// TIA Portal project "taglierina_V15.1" (V15.1)

(* hardware
DEVICE "S71500/ET200MP station_1"  S7-1500 station
   slot 0: "Telaio di montaggio_0"  Rack  6ES7 590-1***0-0AA0
   slot 0: "PM 190W 120/230VAC"  PM 190W 120/230VAC  6EP1333-4BA00
   slot 1: "PLC_1"  CPU 1516-3 PN/DP  6ES7 516-3AN01-0AB0  V2.5
      slot 3: "Display CPU_1"  6ES7591-1BA00-0AA0
   slot 2: "DI 32x24VDC HF_1"  DI 32x24VDC HF  6ES7 521-1BL00-0AB0  V2.0
   slot 3: "DQ 32x24VDC/0.5A HF_1"  DQ 32x24VDC/0.5A HF  6ES7 522-1BL01-0AB0  V1.0
   slot 4: "AI 8xU/I/RTD/TC ST_1"  AI 8xU/I/RTD/TC ST  6ES7 531-7KF00-0AB0  V2.0
   slot 5: "AQ 4xU/I ST_1"  AQ 4xU/I ST  6ES7 532-5HD00-0AB0  V2.0
*)

// ===== PLC "PLC_1"  CPU 1516-3 PN/DP =====

VAR_GLOBAL   // PLC tag table "Tabella delle variabili standard"
   "Clock_Byte" AT %MB100 : Byte;
   "Clock_10Hz" AT %M100.0 : Bool;
   "Clock_5Hz" AT %M100.1 : Bool;
   "Clock_2.5Hz" AT %M100.2 : Bool;
   "Clock_2Hz" AT %M100.3 : Bool;
   "Clock_1.25Hz" AT %M100.4 : Bool;
   "Clock_1Hz" AT %M100.5 : Bool;
   "Clock_0.625Hz" AT %M100.6 : Bool;
   "Clock_0.5Hz" AT %M100.7 : Bool;
   "tmp" AT %M99.0 : Bool;
   "iApriMorsa" AT %I0.0 : Bool;   // Pulsante Morsa aperta
   "iChiudiMorsa" AT %I0.1 : Bool;   // Pulsante Morsa chiusa
   "iAuto" AT %I0.2 : Bool;   // Pulsante Marcia
   "iReset" AT %I0.3 : Bool;   // Pulsante Inizializzazione
   "iStop" AT %I0.4 : Bool;   // Pulsante Stop
   "iIndietro" AT %I0.5 : Bool;   // Taglierina in sede
   "iAvanti" AT %I0.6 : Bool;   // Taglierina Fuori Sede
   "tag_1" AT %I0.7 : Bool;
   "iMorsa2Far" AT %I1.0 : Bool;   // Morsa Mobile Lontana
   "tag_2" AT %I1.1 : Bool;
   "iMorsa1Ch" AT %I1.2 : Bool;   // Morsa Fissa Chiusa (Logica Negata)
   "tag_3" AT %I1.3 : Bool;
   "iMorsa2Ch" AT %I1.4 : Bool;   // Morsa Mobile Chiusa (Logica Negata)
   "iSchermo" AT %I1.5 : Bool;   // Sensore Schermo Sicurezza
   "iEmergenza" AT %I1.6 : Bool;   // Pulsante Emergenza (NC)
   "Tag_16" AT %I1.7 : Bool;
   "Tag_17" AT %I2.0 : Bool;
   "Tag_18" AT %I2.1 : Bool;
   "Tag_19" AT %I2.2 : Bool;
   "Tag_20" AT %I2.3 : Bool;
   "Tag_21" AT %I2.4 : Bool;
   "Tag_22" AT %I2.5 : Bool;
   "Tag_23" AT %I2.6 : Bool;
   "Tag_24" AT %I2.7 : Bool;
   "Tag_25" AT %I3.0 : Bool;
   "Tag_26" AT %I3.1 : Bool;
   "Tag_27" AT %I3.2 : Bool;
   "Tag_28" AT %I3.3 : Bool;
   "Tag_29" AT %I3.5 : Bool;
   "Tag_30" AT %I3.4 : Bool;
   "Tag_31" AT %I3.6 : Bool;
   "Tag_32" AT %I3.7 : Bool;
   "oAvanti" AT %Q0.0 : Bool;   // Spostamento taglierina Fuori Sede (monostabile)
   "oMorsa2Near" AT %Q0.1 : Bool;   // Avvicinamento Morsa Mobile
   "oMorsa2Far" AT %Q0.2 : Bool;   // Allontanamento Morsa Mobile
   "oMorsa1Ch" AT %Q0.3 : Bool;   // Chiusura Morsa Fissa (Monostabile)
   "oMorsa2Ap" AT %Q0.4 : Bool;   // Apertura Morsa Mobile
   "oMorsa2Ch" AT %Q0.5 : Bool;   // Chiusura Morsa Mobile
   "oTaglio" AT %Q0.6 : Bool;   // Motore Taglierina
   "oLedVerde" AT %Q0.7 : Bool;   // Led Verde (da accendere in parallelo al taglio)
   "Tag_41" AT %Q1.0 : Bool;
   "Tag_42" AT %Q1.1 : Bool;
   "Tag_43" AT %Q1.2 : Bool;
   "Tag_44" AT %Q1.3 : Bool;
   "Tag_45" AT %Q1.4 : Bool;
   "Tag_46" AT %Q1.5 : Bool;
   "Tag_47" AT %Q1.6 : Bool;
   "Tag_48" AT %Q1.7 : Bool;
   "Tag_49" AT %Q2.0 : Bool;
   "Tag_50" AT %Q2.1 : Bool;
   "Tag_51" AT %Q2.2 : Bool;
   "Tag_52" AT %Q2.3 : Bool;
   "Tag_53" AT %Q2.4 : Bool;
   "Tag_54" AT %Q2.5 : Bool;
   "Tag_55" AT %Q2.6 : Bool;
   "Tag_56" AT %Q2.7 : Bool;
   "Tag_57" AT %Q3.0 : Bool;
   "Tag_58" AT %Q3.1 : Bool;
   "Tag_59" AT %Q3.2 : Bool;
   "Tag_60" AT %Q3.3 : Bool;
   "Tag_61" AT %Q3.4 : Bool;
   "Tag_62" AT %Q3.5 : Bool;
   "Tag_63" AT %Q3.6 : Bool;
   "Tag_64" AT %Q3.7 : Bool;
END_VAR

VAR_GLOBAL   // PLC tag table "merker"
   "bLamp" AT %M0.0 : Bool;
   "aus" AT %M0.1 : Bool;
   "onsResetCicli" AT %M0.3 : Bool;
   "onsCntCicli" AT %M0.2 : Bool;
END_VAR

DATA_BLOCK "DB_tappe"   // DB1
{ S7_Optimized_Access := 'FALSE' }
VERSION : 0.1
   VAR
      tappeGemma : Array[0..15] of Bool;
      tappeM1 : Array[0..31] of Bool;
      tappeM2 : Array[0..31] of Bool;
      tappeHome : Array[0..15] of Bool;
   END_VAR
BEGIN
END_DATA_BLOCK

DATA_BLOCK "DB_scada"   // DB2
{ S7_Optimized_Access := 'TRUE' }
VERSION : 0.1
   VAR
      scada : Array[0..159] of Bool;
   END_VAR
BEGIN
END_DATA_BLOCK

DATA_BLOCK "DB_comandi"   // DB3
{ S7_Optimized_Access := 'FALSE' }
VERSION : 0.1
   VAR
      bStop : Bool;
      bAuto : Bool;
      bMan : Bool;
      bReset : Bool;
      bEmergenza : Bool;
      free_1 : Bool;
      bAvanti : Bool;   // Comando Spostamento taglierina Fuori Sede (monostabile)
      bMorsa2Near : Bool;   // Comando Avvicinamento Morsa Mobile
      bMorsa2Far : Bool;   // Comando Allontanamento Morsa Mobile
      bMorsa1Ch : Bool;   // Comando Chiusura Morsa Fissa (Monostabile)
      bMorsa2Ap : Bool;   // Comando Apertura Morsa Mobile
      bMorsa2Ch : Bool;   // Comando Chiusura Morsa Mobile
      bTaglio : Bool;   // Comando Motore Taglierina
      bLedVerde : Bool;   // Comando Led Verde (da accednere in parallelo al taglio)
      free_10 : Bool;
      free_11 : Bool;
      free_12 : Bool;
      free_13 : Bool;
      free_14 : Bool;
      free_15 : Bool;
      free_16 : Bool;
      free_17 : Bool;
      free_18 : Bool;
      free_19 : Bool;
      free_20 : Bool;
      free_21 : Bool;
      free_22 : Bool;
      free_23 : Bool;
      free_24 : Bool;
      free_25 : Bool;
      free_26 : Bool;
      xxxxxx : Bool;
   END_VAR
BEGIN
END_DATA_BLOCK

DATA_BLOCK "DB_stati"   // DB4
{ S7_Optimized_Access := 'FALSE' }
VERSION : 0.1
   VAR
      sAuto : Bool;
      sStop : Bool;
      sMan : Bool;
      sHome : Bool;
      sAttesaStop : Bool;
      sEmergenza : Bool;
      xfree : Bool;
      xfree_1 : Bool;
      xfree_2 : Bool;
      xfree_3 : Bool;
      xfree_4 : Bool;
      xfree_5 : Bool;
      xfree_6 : Bool;
      xfree_7 : Bool;
      xfree_8 : Bool;
      xfree_9 : Bool;
      bIni1 : Bool;
      bIni2 : Bool;
      bRip1 : Bool;
      bRip2 : Bool;
      free1 : Bool;
      free2 : Bool;
      free3 : Bool;
      free4 : Bool;
      free5 : Bool;
      free6 : Bool;
      free7 : Bool;
      free8 : Bool;
      free9 : Bool;
      free10 : Bool;
      free11 : Bool;
      free12 : Bool;
   END_VAR
BEGIN
END_DATA_BLOCK

DATA_BLOCK "DB_parametriInt"   // DB5
{ S7_Optimized_Access := 'FALSE' }
VERSION : 0.1
   VAR
      cntCicli : Int := 0;
      free1 : Int;
      free2 : Int;
      free3 : Int;
      free4 : Int;
      free5 : Int;
      free6 : Int;
      free7 : Int;
   END_VAR
BEGIN
END_DATA_BLOCK

DATA_BLOCK "DB_scadaInt"   // DB6
{ S7_Optimized_Access := 'TRUE' }
VERSION : 0.1
   VAR
      scadaInt : Array[0..7] of Int;
   END_VAR
BEGIN
END_DATA_BLOCK

// folder: System blocks/Program resources

DATA_BLOCK "tResetPulsanti"   // DB7
{ S7_Optimized_Access := 'TRUE' }
AUTHOR : Simatic
FAMILY : IEC
NAME : IEC_TMR
VERSION : 1.0
// stored: InstanceOfName IEC_TIMER
"IEC_TIMER"
BEGIN
END_DATA_BLOCK

// folder: (top level)

FUNCTION "_resetPulsanti" : Void   // FC1, LAD
{ S7_Optimized_Access := 'TRUE' }
VERSION : 0.1
BEGIN

REGION Network 1
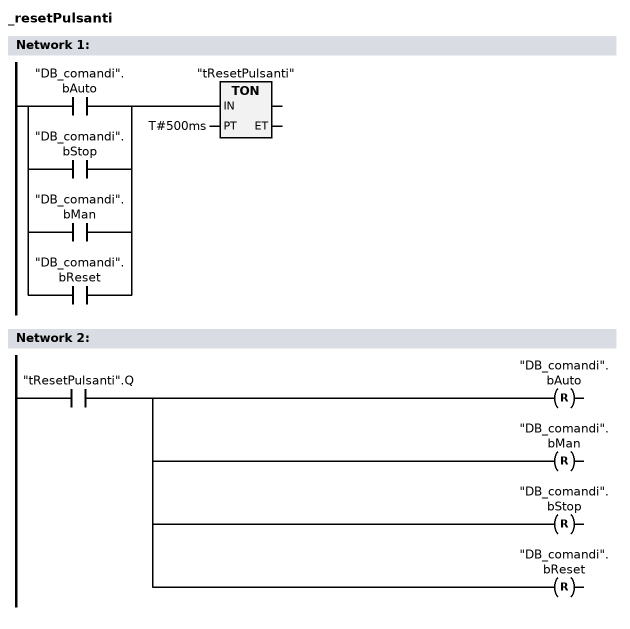
   "tResetPulsanti".TON(IN := "DB_comandi".bAuto OR "DB_comandi".bStop OR "DB_comandi".bMan OR "DB_comandi".bReset,
                        PT := T#500ms);
END_REGION

REGION Network 2
   RUNG wire#powerrail
      Contact( "tResetPulsanti".Q )
      wire#w1
      R_Coil( "DB_comandi".bAuto )
   END_RUNG
   RUNG wire#w1
      R_Coil( "DB_comandi".bMan )
   END_RUNG
   RUNG wire#w1
      R_Coil( "DB_comandi".bStop )
   END_RUNG
   RUNG wire#w1
      R_Coil( "DB_comandi".bReset )
   END_RUNG
   // the same network as SCL:
   IF "tResetPulsanti".Q THEN
       "DB_comandi".bAuto := FALSE;
       "DB_comandi".bMan := FALSE;
       "DB_comandi".bStop := FALSE;
       "DB_comandi".bReset := FALSE;
   END_IF;
END_REGION
END_FUNCTION

FUNCTION "_lampeggio" : Void   // FC2, LAD
{ S7_Optimized_Access := 'TRUE' }
VERSION : 0.1
BEGIN

REGION Network 1
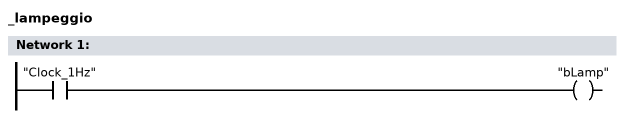
   RUNG wire#powerrail
      Contact( "Clock_1Hz" )
      Coil( "bLamp" )
   END_RUNG
   // the same network as SCL:
   "bLamp" := "Clock_1Hz";
END_REGION
END_FUNCTION

FUNCTION "_gemma" : Void   // FC3, LAD
{ S7_Optimized_Access := 'TRUE' }
VERSION : 0.1
   VAR_TEMP   // added for the SCL form of the ladder/FBD networks
      _w1 : Bool;
   END_VAR
BEGIN

REGION Network 1
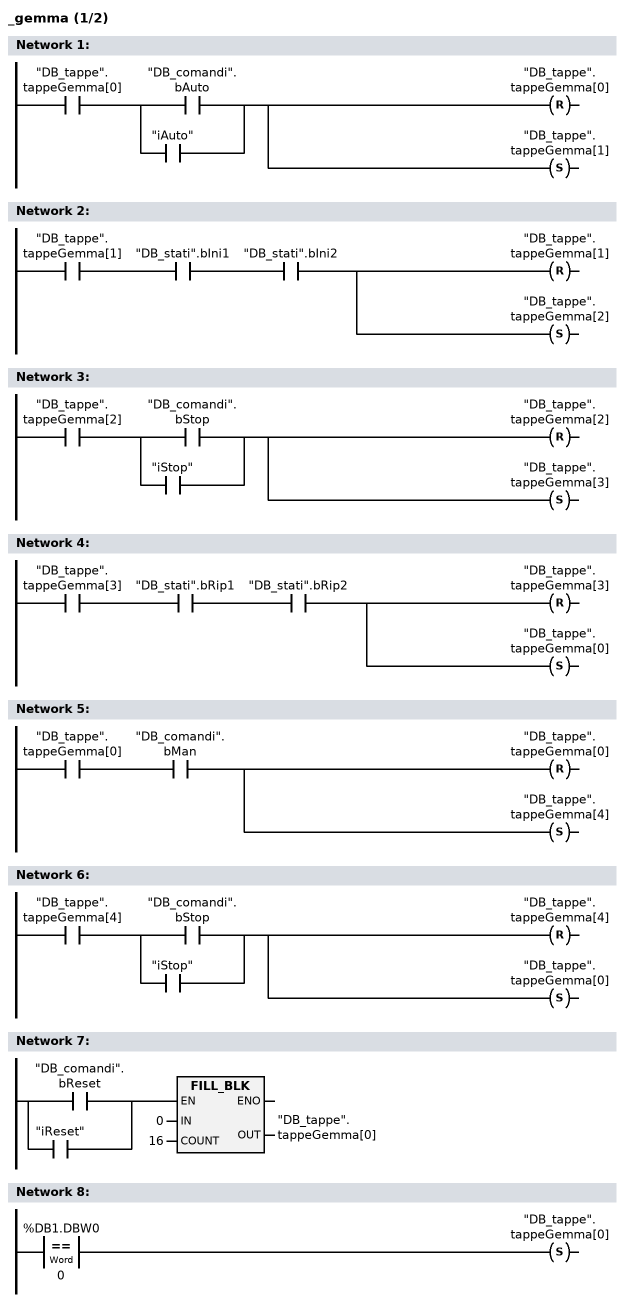
   RUNG wire#powerrail
      Contact( "DB_tappe".tappeGemma[0] )
      wire#w1
      Contact( "DB_comandi".bAuto )
      wire#w2
      R_Coil( "DB_tappe".tappeGemma[0] )
   END_RUNG
   RUNG wire#w1
      Contact( "iAuto" )
   END_RUNG wire#w2
   RUNG wire#w2
      S_Coil( "DB_tappe".tappeGemma[1] )
   END_RUNG
   // the same network as SCL:
   #_w1 := "DB_tappe".tappeGemma[0] AND ("DB_comandi".bAuto OR "iAuto");
   IF #_w1 THEN
       "DB_tappe".tappeGemma[0] := FALSE;
       "DB_tappe".tappeGemma[1] := TRUE;
   END_IF;
END_REGION

REGION Network 2
   RUNG wire#powerrail
      Contact( "DB_tappe".tappeGemma[1] )
      Contact( "DB_stati".bIni1 )
      Contact( "DB_stati".bIni2 )
      wire#w1
      R_Coil( "DB_tappe".tappeGemma[1] )
   END_RUNG
   RUNG wire#w1
      S_Coil( "DB_tappe".tappeGemma[2] )
   END_RUNG
   // the same network as SCL:
   #_w1 := "DB_tappe".tappeGemma[1] AND "DB_stati".bIni1 AND "DB_stati".bIni2;
   IF #_w1 THEN
       "DB_tappe".tappeGemma[1] := FALSE;
       "DB_tappe".tappeGemma[2] := TRUE;
   END_IF;
END_REGION

REGION Network 3
   RUNG wire#powerrail
      Contact( "DB_tappe".tappeGemma[2] )
      wire#w1
      Contact( "DB_comandi".bStop )
      wire#w2
      R_Coil( "DB_tappe".tappeGemma[2] )
   END_RUNG
   RUNG wire#w1
      Contact( "iStop" )
   END_RUNG wire#w2
   RUNG wire#w2
      S_Coil( "DB_tappe".tappeGemma[3] )
   END_RUNG
   // the same network as SCL:
   #_w1 := "DB_tappe".tappeGemma[2] AND ("DB_comandi".bStop OR "iStop");
   IF #_w1 THEN
       "DB_tappe".tappeGemma[2] := FALSE;
       "DB_tappe".tappeGemma[3] := TRUE;
   END_IF;
END_REGION

REGION Network 4
   RUNG wire#powerrail
      Contact( "DB_tappe".tappeGemma[3] )
      Contact( "DB_stati".bRip1 )
      Contact( "DB_stati".bRip2 )
      wire#w1
      R_Coil( "DB_tappe".tappeGemma[3] )
   END_RUNG
   RUNG wire#w1
      S_Coil( "DB_tappe".tappeGemma[0] )
   END_RUNG
   // the same network as SCL:
   #_w1 := "DB_tappe".tappeGemma[3] AND "DB_stati".bRip1 AND "DB_stati".bRip2;
   IF #_w1 THEN
       "DB_tappe".tappeGemma[3] := FALSE;
       "DB_tappe".tappeGemma[0] := TRUE;
   END_IF;
END_REGION

REGION Network 5
   RUNG wire#powerrail
      Contact( "DB_tappe".tappeGemma[0] )
      Contact( "DB_comandi".bMan )
      wire#w1
      R_Coil( "DB_tappe".tappeGemma[0] )
   END_RUNG
   RUNG wire#w1
      S_Coil( "DB_tappe".tappeGemma[4] )
   END_RUNG
   // the same network as SCL:
   #_w1 := "DB_tappe".tappeGemma[0] AND "DB_comandi".bMan;
   IF #_w1 THEN
       "DB_tappe".tappeGemma[0] := FALSE;
       "DB_tappe".tappeGemma[4] := TRUE;
   END_IF;
END_REGION

REGION Network 6
   RUNG wire#powerrail
      Contact( "DB_tappe".tappeGemma[4] )
      wire#w1
      Contact( "DB_comandi".bStop )
      wire#w2
      R_Coil( "DB_tappe".tappeGemma[4] )
   END_RUNG
   RUNG wire#w1
      Contact( "iStop" )
   END_RUNG wire#w2
   RUNG wire#w2
      S_Coil( "DB_tappe".tappeGemma[0] )
   END_RUNG
   // the same network as SCL:
   #_w1 := "DB_tappe".tappeGemma[4] AND ("DB_comandi".bStop OR "iStop");
   IF #_w1 THEN
       "DB_tappe".tappeGemma[4] := FALSE;
       "DB_tappe".tappeGemma[0] := TRUE;
   END_IF;
END_REGION

REGION Network 7
   RUNG wire#powerrail
      Contact( "DB_comandi".bReset )
      wire#w1
      FillBlockI(in := 0, count := 16, out => "DB_tappe".tappeGemma[0])
   END_RUNG
   RUNG wire#powerrail
      Contact( "iReset" )
   END_RUNG wire#w1
   // the same network as SCL:
   IF "DB_comandi".bReset OR "iReset" THEN
       FILL_BLK(IN := 0, COUNT := 16, OUT => "DB_tappe".tappeGemma[0]);
   END_IF;
END_REGION

REGION Network 8
   RUNG wire#powerrail
      { S7_Templates := "SrcType := Word" } EQ_Contact(in1 := %DB1.DBW0, in2 := 0)
      S_Coil( "DB_tappe".tappeGemma[0] )
   END_RUNG
   // the same network as SCL:
   IF %DB1.DBW0 = 0 THEN "DB_tappe".tappeGemma[0] := TRUE; END_IF;
END_REGION

REGION Network 9
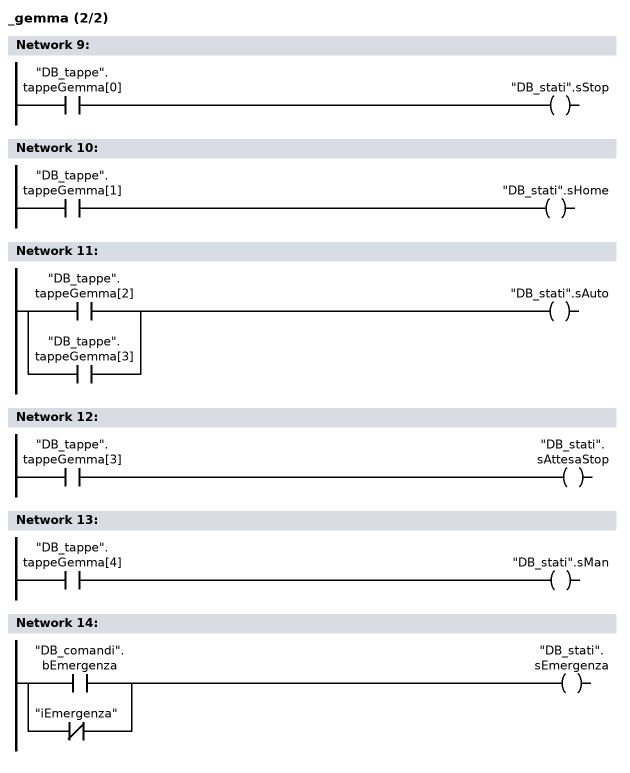
   RUNG wire#powerrail
      Contact( "DB_tappe".tappeGemma[0] )
      Coil( "DB_stati".sStop )
   END_RUNG
   // the same network as SCL:
   "DB_stati".sStop := "DB_tappe".tappeGemma[0];
END_REGION

REGION Network 10
   RUNG wire#powerrail
      Contact( "DB_tappe".tappeGemma[1] )
      Coil( "DB_stati".sHome )
   END_RUNG
   // the same network as SCL:
   "DB_stati".sHome := "DB_tappe".tappeGemma[1];
END_REGION

REGION Network 11
   RUNG wire#powerrail
      Contact( "DB_tappe".tappeGemma[2] )
      wire#w1
      Coil( "DB_stati".sAuto )
   END_RUNG
   RUNG wire#powerrail
      Contact( "DB_tappe".tappeGemma[3] )
   END_RUNG wire#w1
   // the same network as SCL:
   "DB_stati".sAuto := "DB_tappe".tappeGemma[2] OR "DB_tappe".tappeGemma[3];
END_REGION

REGION Network 12
   RUNG wire#powerrail
      Contact( "DB_tappe".tappeGemma[3] )
      Coil( "DB_stati".sAttesaStop )
   END_RUNG
   // the same network as SCL:
   "DB_stati".sAttesaStop := "DB_tappe".tappeGemma[3];
END_REGION

REGION Network 13
   RUNG wire#powerrail
      Contact( "DB_tappe".tappeGemma[4] )
      Coil( "DB_stati".sMan )
   END_RUNG
   // the same network as SCL:
   "DB_stati".sMan := "DB_tappe".tappeGemma[4];
END_REGION

REGION Network 14
   RUNG wire#powerrail
      Contact( "DB_comandi".bEmergenza )
      wire#w1
      Coil( "DB_stati".sEmergenza )
   END_RUNG
   RUNG wire#powerrail
      I_Contact( "iEmergenza" )
   END_RUNG wire#w1
   // the same network as SCL:
   "DB_stati".sEmergenza := "DB_comandi".bEmergenza OR NOT "iEmergenza";
END_REGION
END_FUNCTION

FUNCTION "_grafcet_M1" : Void   // FC4, LAD
{ S7_Optimized_Access := 'TRUE' }
VERSION : 0.1
   VAR_TEMP   // added for the SCL form of the ladder/FBD networks
      _w1 : Bool;
   END_VAR
BEGIN

REGION Network 1: ***************************************************************************************
   // ************************  ISTRUZIONI DI RESET ***********************************
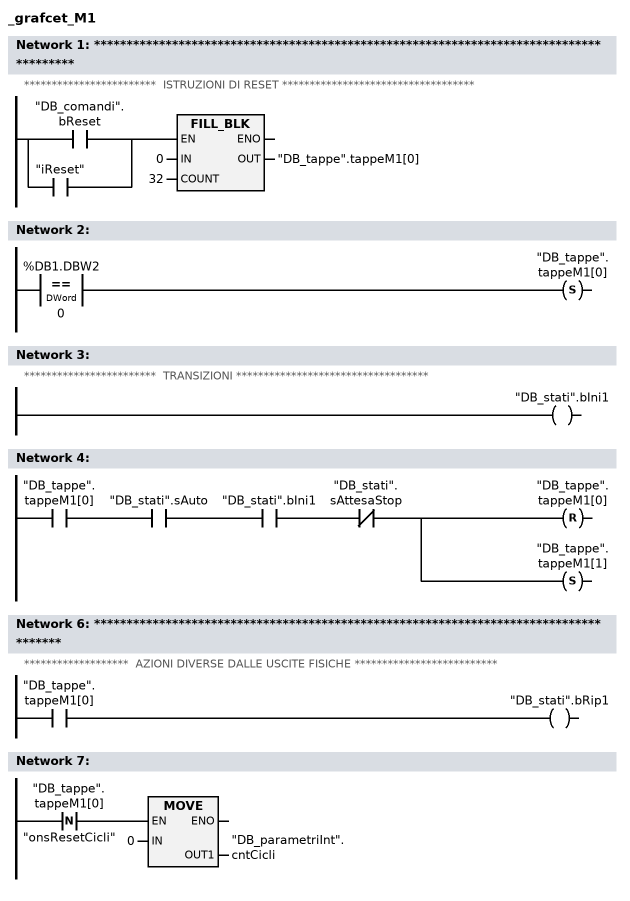
   RUNG wire#powerrail
      Contact( "DB_comandi".bReset )
      wire#w1
      FillBlockI(in := 0, count := 32, out => "DB_tappe".tappeM1[0])
   END_RUNG
   RUNG wire#powerrail
      Contact( "iReset" )
   END_RUNG wire#w1
   // the same network as SCL:
   IF "DB_comandi".bReset OR "iReset" THEN
       FILL_BLK(IN := 0, COUNT := 32, OUT => "DB_tappe".tappeM1[0]);
   END_IF;
END_REGION

REGION Network 2
   RUNG wire#powerrail
      { S7_Templates := "SrcType := DWord" } EQ_Contact(in1 := %DB1.DBW2, in2 := 0)
      S_Coil( "DB_tappe".tappeM1[0] )
   END_RUNG
   // the same network as SCL:
   IF %DB1.DBW2 = 0 THEN "DB_tappe".tappeM1[0] := TRUE; END_IF;
END_REGION

REGION Network 3
   // ************************  TRANSIZIONI ***********************************
   RUNG wire#powerrail
      Coil( "DB_stati".bIni1 )
   END_RUNG
   // the same network as SCL:
   "DB_stati".bIni1 := TRUE;
END_REGION

REGION Network 4
   RUNG wire#powerrail
      Contact( "DB_tappe".tappeM1[0] )
      Contact( "DB_stati".sAuto )
      Contact( "DB_stati".bIni1 )
      I_Contact( "DB_stati".sAttesaStop )
      wire#w1
      R_Coil( "DB_tappe".tappeM1[0] )
   END_RUNG
   RUNG wire#w1
      S_Coil( "DB_tappe".tappeM1[1] )
   END_RUNG
   // the same network as SCL:
   #_w1 := "DB_tappe".tappeM1[0] AND "DB_stati".sAuto AND "DB_stati".bIni1 AND NOT "DB_stati".sAttesaStop;
   IF #_w1 THEN
       "DB_tappe".tappeM1[0] := FALSE;
       "DB_tappe".tappeM1[1] := TRUE;
   END_IF;
END_REGION

REGION Network 6: *************************************************************************************
   // *******************  AZIONI DIVERSE DALLE USCITE FISICHE **************************
   RUNG wire#powerrail
      Contact( "DB_tappe".tappeM1[0] )
      Coil( "DB_stati".bRip1 )
   END_RUNG
   // the same network as SCL:
   "DB_stati".bRip1 := "DB_tappe".tappeM1[0];
END_REGION

REGION Network 7
   RUNG wire#powerrail
      N_Contact(operand := "DB_tappe".tappeM1[0], bit := "onsResetCicli")
      Move(in := 0, out1 => "DB_parametriInt".cntCicli)
   END_RUNG
   // the same network as SCL:
   #_w1 := NOT "DB_tappe".tappeM1[0] AND "onsResetCicli";   // falling edge of "DB_tappe".tappeM1[0]
   "onsResetCicli" := "DB_tappe".tappeM1[0];
   IF #_w1 THEN "DB_parametriInt".cntCicli := 0; END_IF;
END_REGION
END_FUNCTION

FUNCTION "_grafcet_M2" : Void   // FC5, LAD
{ S7_Optimized_Access := 'TRUE' }
VERSION : 0.1
   VAR_TEMP   // added for the SCL form of the ladder/FBD networks
      _w1 : Bool;
   END_VAR
BEGIN

REGION Network 1: ***************************************************************************************
   // ************************  ISTRUZIONI DI RESET ***********************************
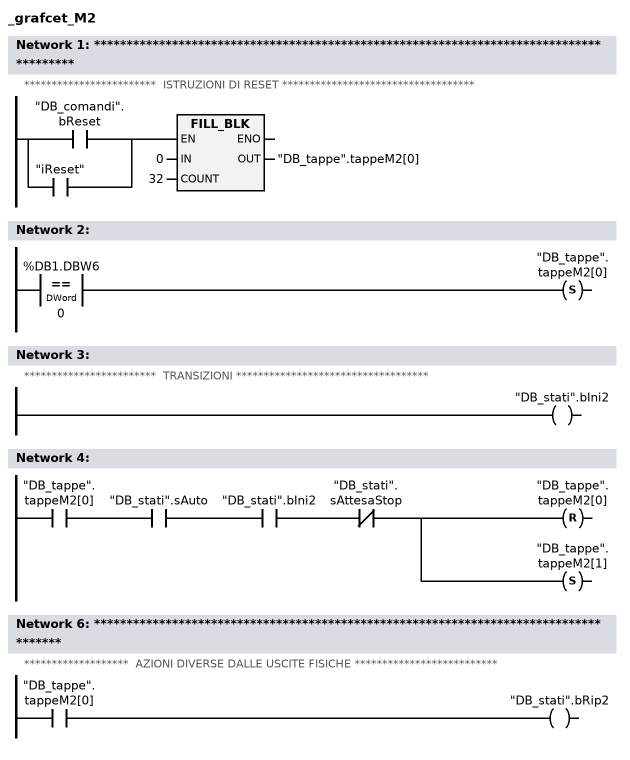
   RUNG wire#powerrail
      Contact( "DB_comandi".bReset )
      wire#w1
      FillBlockI(in := 0, count := 32, out => "DB_tappe".tappeM2[0])
   END_RUNG
   RUNG wire#powerrail
      Contact( "iReset" )
   END_RUNG wire#w1
   // the same network as SCL:
   IF "DB_comandi".bReset OR "iReset" THEN
       FILL_BLK(IN := 0, COUNT := 32, OUT => "DB_tappe".tappeM2[0]);
   END_IF;
END_REGION

REGION Network 2
   RUNG wire#powerrail
      { S7_Templates := "SrcType := DWord" } EQ_Contact(in1 := %DB1.DBW6, in2 := 0)
      S_Coil( "DB_tappe".tappeM2[0] )
   END_RUNG
   // the same network as SCL:
   IF %DB1.DBW6 = 0 THEN "DB_tappe".tappeM2[0] := TRUE; END_IF;
END_REGION

REGION Network 3
   // ************************  TRANSIZIONI ***********************************
   RUNG wire#powerrail
      Coil( "DB_stati".bIni2 )
   END_RUNG
   // the same network as SCL:
   "DB_stati".bIni2 := TRUE;
END_REGION

REGION Network 4
   RUNG wire#powerrail
      Contact( "DB_tappe".tappeM2[0] )
      Contact( "DB_stati".sAuto )
      Contact( "DB_stati".bIni2 )
      I_Contact( "DB_stati".sAttesaStop )
      wire#w1
      R_Coil( "DB_tappe".tappeM2[0] )
   END_RUNG
   RUNG wire#w1
      S_Coil( "DB_tappe".tappeM2[1] )
   END_RUNG
   // the same network as SCL:
   #_w1 := "DB_tappe".tappeM2[0] AND "DB_stati".sAuto AND "DB_stati".bIni2 AND NOT "DB_stati".sAttesaStop;
   IF #_w1 THEN
       "DB_tappe".tappeM2[0] := FALSE;
       "DB_tappe".tappeM2[1] := TRUE;
   END_IF;
END_REGION

REGION Network 6: *************************************************************************************
   // *******************  AZIONI DIVERSE DALLE USCITE FISICHE **************************
   RUNG wire#powerrail
      Contact( "DB_tappe".tappeM2[0] )
      Coil( "DB_stati".bRip2 )
   END_RUNG
   // the same network as SCL:
   "DB_stati".bRip2 := "DB_tappe".tappeM2[0];
END_REGION
END_FUNCTION

FUNCTION "_uscite" : Void   // FC6, LAD
{ S7_Optimized_Access := 'TRUE' }
VERSION : 0.1
BEGIN

REGION Network 1
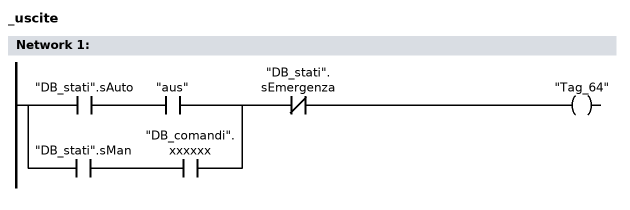
   RUNG wire#powerrail
      Contact( "DB_stati".sAuto )
      Contact( "aus" )
      wire#w1
      I_Contact( "DB_stati".sEmergenza )
      Coil( "Tag_64" )
   END_RUNG
   RUNG wire#powerrail
      Contact( "DB_stati".sMan )
      Contact( "DB_comandi".xxxxxx )
   END_RUNG wire#w1
   // the same network as SCL:
   "Tag_64" := (("DB_stati".sAuto AND "aus") OR ("DB_stati".sMan AND "DB_comandi".xxxxxx)) AND NOT "DB_stati".sEmergenza;
END_REGION
END_FUNCTION

FUNCTION "_scada" : Void   // FC8, LAD
{ S7_Optimized_Access := 'TRUE' }
VERSION : 0.1
BEGIN

REGION Network 1
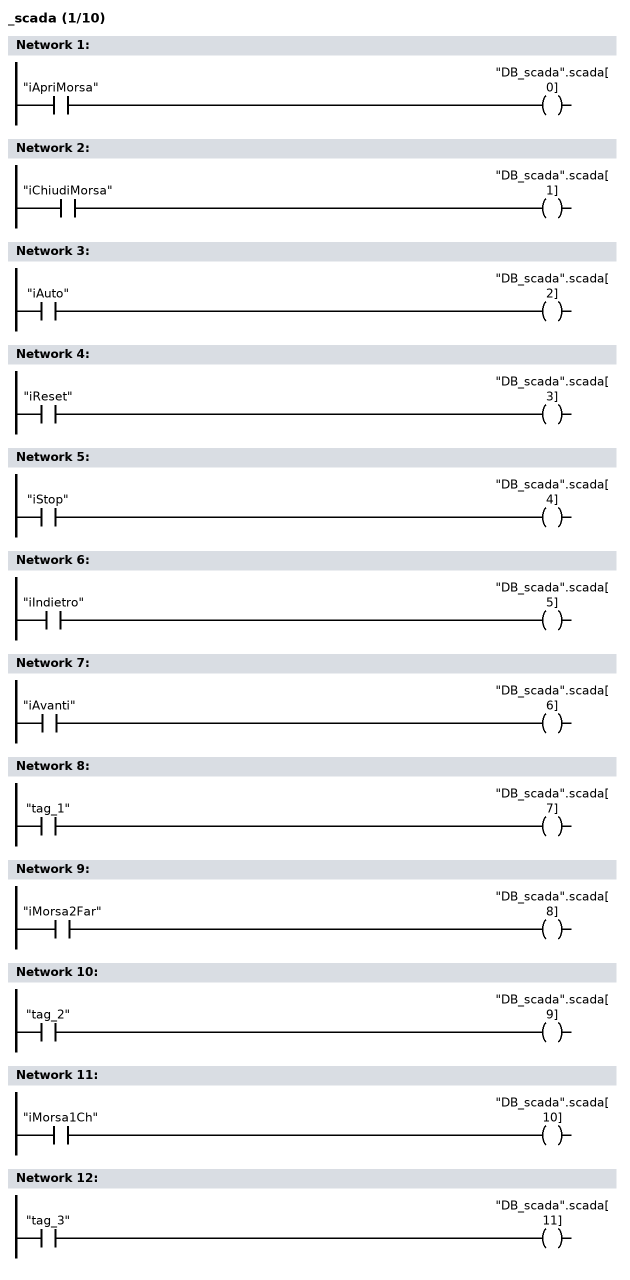
   RUNG wire#powerrail
      Contact( "iApriMorsa" )
      Coil( "DB_scada".scada[0] )
   END_RUNG
   // the same network as SCL:
   "DB_scada".scada[0] := "iApriMorsa";
END_REGION

REGION Network 2
   RUNG wire#powerrail
      Contact( "iChiudiMorsa" )
      Coil( "DB_scada".scada[1] )
   END_RUNG
   // the same network as SCL:
   "DB_scada".scada[1] := "iChiudiMorsa";
END_REGION

REGION Network 3
   RUNG wire#powerrail
      Contact( "iAuto" )
      Coil( "DB_scada".scada[2] )
   END_RUNG
   // the same network as SCL:
   "DB_scada".scada[2] := "iAuto";
END_REGION

REGION Network 4
   RUNG wire#powerrail
      Contact( "iReset" )
      Coil( "DB_scada".scada[3] )
   END_RUNG
   // the same network as SCL:
   "DB_scada".scada[3] := "iReset";
END_REGION

REGION Network 5
   RUNG wire#powerrail
      Contact( "iStop" )
      Coil( "DB_scada".scada[4] )
   END_RUNG
   // the same network as SCL:
   "DB_scada".scada[4] := "iStop";
END_REGION

REGION Network 6
   RUNG wire#powerrail
      Contact( "iIndietro" )
      Coil( "DB_scada".scada[5] )
   END_RUNG
   // the same network as SCL:
   "DB_scada".scada[5] := "iIndietro";
END_REGION

REGION Network 7
   RUNG wire#powerrail
      Contact( "iAvanti" )
      Coil( "DB_scada".scada[6] )
   END_RUNG
   // the same network as SCL:
   "DB_scada".scada[6] := "iAvanti";
END_REGION

REGION Network 8
   RUNG wire#powerrail
      Contact( "tag_1" )
      Coil( "DB_scada".scada[7] )
   END_RUNG
   // the same network as SCL:
   "DB_scada".scada[7] := "tag_1";
END_REGION

REGION Network 9
   RUNG wire#powerrail
      Contact( "iMorsa2Far" )
      Coil( "DB_scada".scada[8] )
   END_RUNG
   // the same network as SCL:
   "DB_scada".scada[8] := "iMorsa2Far";
END_REGION

REGION Network 10
   RUNG wire#powerrail
      Contact( "tag_2" )
      Coil( "DB_scada".scada[9] )
   END_RUNG
   // the same network as SCL:
   "DB_scada".scada[9] := "tag_2";
END_REGION

REGION Network 11
   RUNG wire#powerrail
      Contact( "iMorsa1Ch" )
      Coil( "DB_scada".scada[10] )
   END_RUNG
   // the same network as SCL:
   "DB_scada".scada[10] := "iMorsa1Ch";
END_REGION

REGION Network 12
   RUNG wire#powerrail
      Contact( "tag_3" )
      Coil( "DB_scada".scada[11] )
   END_RUNG
   // the same network as SCL:
   "DB_scada".scada[11] := "tag_3";
END_REGION

REGION Network 13
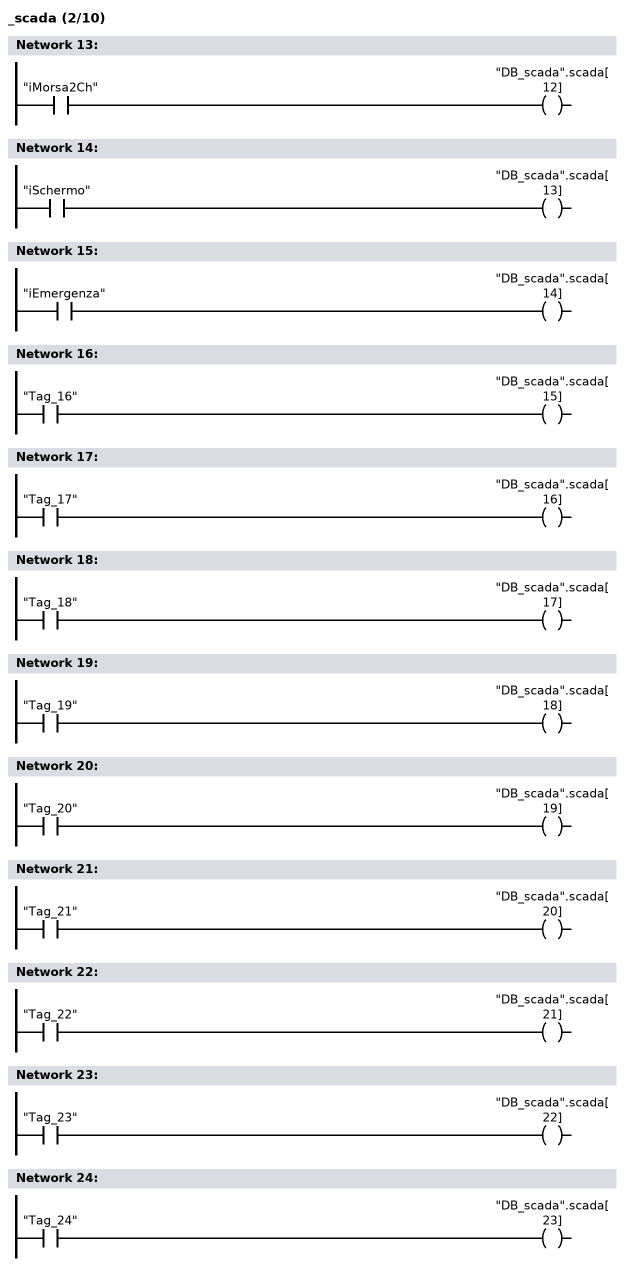
   RUNG wire#powerrail
      Contact( "iMorsa2Ch" )
      Coil( "DB_scada".scada[12] )
   END_RUNG
   // the same network as SCL:
   "DB_scada".scada[12] := "iMorsa2Ch";
END_REGION

REGION Network 14
   RUNG wire#powerrail
      Contact( "iSchermo" )
      Coil( "DB_scada".scada[13] )
   END_RUNG
   // the same network as SCL:
   "DB_scada".scada[13] := "iSchermo";
END_REGION

REGION Network 15
   RUNG wire#powerrail
      Contact( "iEmergenza" )
      Coil( "DB_scada".scada[14] )
   END_RUNG
   // the same network as SCL:
   "DB_scada".scada[14] := "iEmergenza";
END_REGION

REGION Network 16
   RUNG wire#powerrail
      Contact( "Tag_16" )
      Coil( "DB_scada".scada[15] )
   END_RUNG
   // the same network as SCL:
   "DB_scada".scada[15] := "Tag_16";
END_REGION

REGION Network 17
   RUNG wire#powerrail
      Contact( "Tag_17" )
      Coil( "DB_scada".scada[16] )
   END_RUNG
   // the same network as SCL:
   "DB_scada".scada[16] := "Tag_17";
END_REGION

REGION Network 18
   RUNG wire#powerrail
      Contact( "Tag_18" )
      Coil( "DB_scada".scada[17] )
   END_RUNG
   // the same network as SCL:
   "DB_scada".scada[17] := "Tag_18";
END_REGION

REGION Network 19
   RUNG wire#powerrail
      Contact( "Tag_19" )
      Coil( "DB_scada".scada[18] )
   END_RUNG
   // the same network as SCL:
   "DB_scada".scada[18] := "Tag_19";
END_REGION

REGION Network 20
   RUNG wire#powerrail
      Contact( "Tag_20" )
      Coil( "DB_scada".scada[19] )
   END_RUNG
   // the same network as SCL:
   "DB_scada".scada[19] := "Tag_20";
END_REGION

REGION Network 21
   RUNG wire#powerrail
      Contact( "Tag_21" )
      Coil( "DB_scada".scada[20] )
   END_RUNG
   // the same network as SCL:
   "DB_scada".scada[20] := "Tag_21";
END_REGION

REGION Network 22
   RUNG wire#powerrail
      Contact( "Tag_22" )
      Coil( "DB_scada".scada[21] )
   END_RUNG
   // the same network as SCL:
   "DB_scada".scada[21] := "Tag_22";
END_REGION

REGION Network 23
   RUNG wire#powerrail
      Contact( "Tag_23" )
      Coil( "DB_scada".scada[22] )
   END_RUNG
   // the same network as SCL:
   "DB_scada".scada[22] := "Tag_23";
END_REGION

REGION Network 24
   RUNG wire#powerrail
      Contact( "Tag_24" )
      Coil( "DB_scada".scada[23] )
   END_RUNG
   // the same network as SCL:
   "DB_scada".scada[23] := "Tag_24";
END_REGION

REGION Network 25
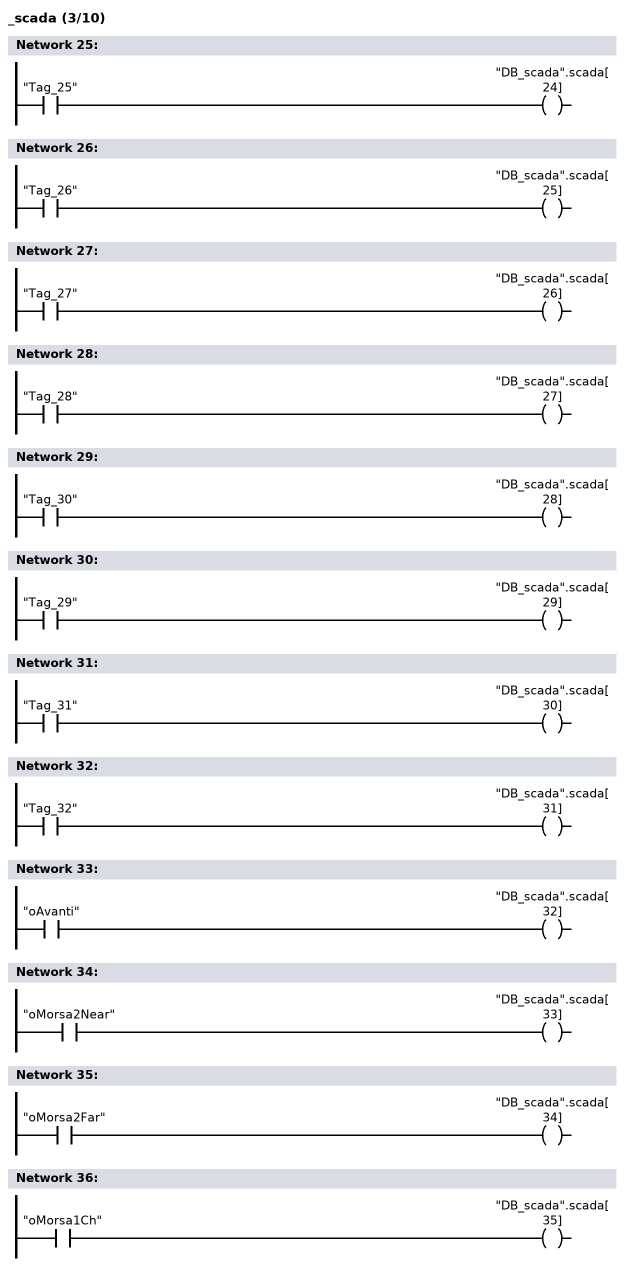
   RUNG wire#powerrail
      Contact( "Tag_25" )
      Coil( "DB_scada".scada[24] )
   END_RUNG
   // the same network as SCL:
   "DB_scada".scada[24] := "Tag_25";
END_REGION

REGION Network 26
   RUNG wire#powerrail
      Contact( "Tag_26" )
      Coil( "DB_scada".scada[25] )
   END_RUNG
   // the same network as SCL:
   "DB_scada".scada[25] := "Tag_26";
END_REGION

REGION Network 27
   RUNG wire#powerrail
      Contact( "Tag_27" )
      Coil( "DB_scada".scada[26] )
   END_RUNG
   // the same network as SCL:
   "DB_scada".scada[26] := "Tag_27";
END_REGION

REGION Network 28
   RUNG wire#powerrail
      Contact( "Tag_28" )
      Coil( "DB_scada".scada[27] )
   END_RUNG
   // the same network as SCL:
   "DB_scada".scada[27] := "Tag_28";
END_REGION

REGION Network 29
   RUNG wire#powerrail
      Contact( "Tag_30" )
      Coil( "DB_scada".scada[28] )
   END_RUNG
   // the same network as SCL:
   "DB_scada".scada[28] := "Tag_30";
END_REGION

REGION Network 30
   RUNG wire#powerrail
      Contact( "Tag_29" )
      Coil( "DB_scada".scada[29] )
   END_RUNG
   // the same network as SCL:
   "DB_scada".scada[29] := "Tag_29";
END_REGION

REGION Network 31
   RUNG wire#powerrail
      Contact( "Tag_31" )
      Coil( "DB_scada".scada[30] )
   END_RUNG
   // the same network as SCL:
   "DB_scada".scada[30] := "Tag_31";
END_REGION

REGION Network 32
   RUNG wire#powerrail
      Contact( "Tag_32" )
      Coil( "DB_scada".scada[31] )
   END_RUNG
   // the same network as SCL:
   "DB_scada".scada[31] := "Tag_32";
END_REGION

REGION Network 33
   RUNG wire#powerrail
      Contact( "oAvanti" )
      Coil( "DB_scada".scada[32] )
   END_RUNG
   // the same network as SCL:
   "DB_scada".scada[32] := "oAvanti";
END_REGION

REGION Network 34
   RUNG wire#powerrail
      Contact( "oMorsa2Near" )
      Coil( "DB_scada".scada[33] )
   END_RUNG
   // the same network as SCL:
   "DB_scada".scada[33] := "oMorsa2Near";
END_REGION

REGION Network 35
   RUNG wire#powerrail
      Contact( "oMorsa2Far" )
      Coil( "DB_scada".scada[34] )
   END_RUNG
   // the same network as SCL:
   "DB_scada".scada[34] := "oMorsa2Far";
END_REGION

REGION Network 36
   RUNG wire#powerrail
      Contact( "oMorsa1Ch" )
      Coil( "DB_scada".scada[35] )
   END_RUNG
   // the same network as SCL:
   "DB_scada".scada[35] := "oMorsa1Ch";
END_REGION

REGION Network 37
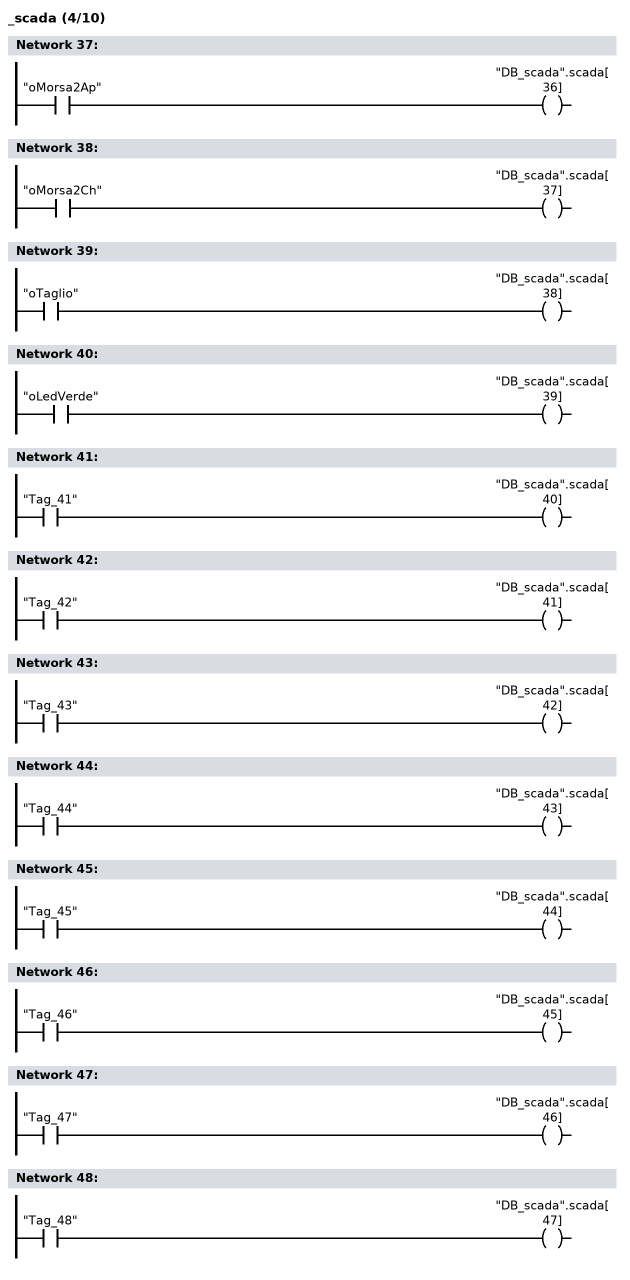
   RUNG wire#powerrail
      Contact( "oMorsa2Ap" )
      Coil( "DB_scada".scada[36] )
   END_RUNG
   // the same network as SCL:
   "DB_scada".scada[36] := "oMorsa2Ap";
END_REGION

REGION Network 38
   RUNG wire#powerrail
      Contact( "oMorsa2Ch" )
      Coil( "DB_scada".scada[37] )
   END_RUNG
   // the same network as SCL:
   "DB_scada".scada[37] := "oMorsa2Ch";
END_REGION

REGION Network 39
   RUNG wire#powerrail
      Contact( "oTaglio" )
      Coil( "DB_scada".scada[38] )
   END_RUNG
   // the same network as SCL:
   "DB_scada".scada[38] := "oTaglio";
END_REGION

REGION Network 40
   RUNG wire#powerrail
      Contact( "oLedVerde" )
      Coil( "DB_scada".scada[39] )
   END_RUNG
   // the same network as SCL:
   "DB_scada".scada[39] := "oLedVerde";
END_REGION

REGION Network 41
   RUNG wire#powerrail
      Contact( "Tag_41" )
      Coil( "DB_scada".scada[40] )
   END_RUNG
   // the same network as SCL:
   "DB_scada".scada[40] := "Tag_41";
END_REGION

REGION Network 42
   RUNG wire#powerrail
      Contact( "Tag_42" )
      Coil( "DB_scada".scada[41] )
   END_RUNG
   // the same network as SCL:
   "DB_scada".scada[41] := "Tag_42";
END_REGION

REGION Network 43
   RUNG wire#powerrail
      Contact( "Tag_43" )
      Coil( "DB_scada".scada[42] )
   END_RUNG
   // the same network as SCL:
   "DB_scada".scada[42] := "Tag_43";
END_REGION

REGION Network 44
   RUNG wire#powerrail
      Contact( "Tag_44" )
      Coil( "DB_scada".scada[43] )
   END_RUNG
   // the same network as SCL:
   "DB_scada".scada[43] := "Tag_44";
END_REGION

REGION Network 45
   RUNG wire#powerrail
      Contact( "Tag_45" )
      Coil( "DB_scada".scada[44] )
   END_RUNG
   // the same network as SCL:
   "DB_scada".scada[44] := "Tag_45";
END_REGION

REGION Network 46
   RUNG wire#powerrail
      Contact( "Tag_46" )
      Coil( "DB_scada".scada[45] )
   END_RUNG
   // the same network as SCL:
   "DB_scada".scada[45] := "Tag_46";
END_REGION

REGION Network 47
   RUNG wire#powerrail
      Contact( "Tag_47" )
      Coil( "DB_scada".scada[46] )
   END_RUNG
   // the same network as SCL:
   "DB_scada".scada[46] := "Tag_47";
END_REGION

REGION Network 48
   RUNG wire#powerrail
      Contact( "Tag_48" )
      Coil( "DB_scada".scada[47] )
   END_RUNG
   // the same network as SCL:
   "DB_scada".scada[47] := "Tag_48";
END_REGION

REGION Network 49
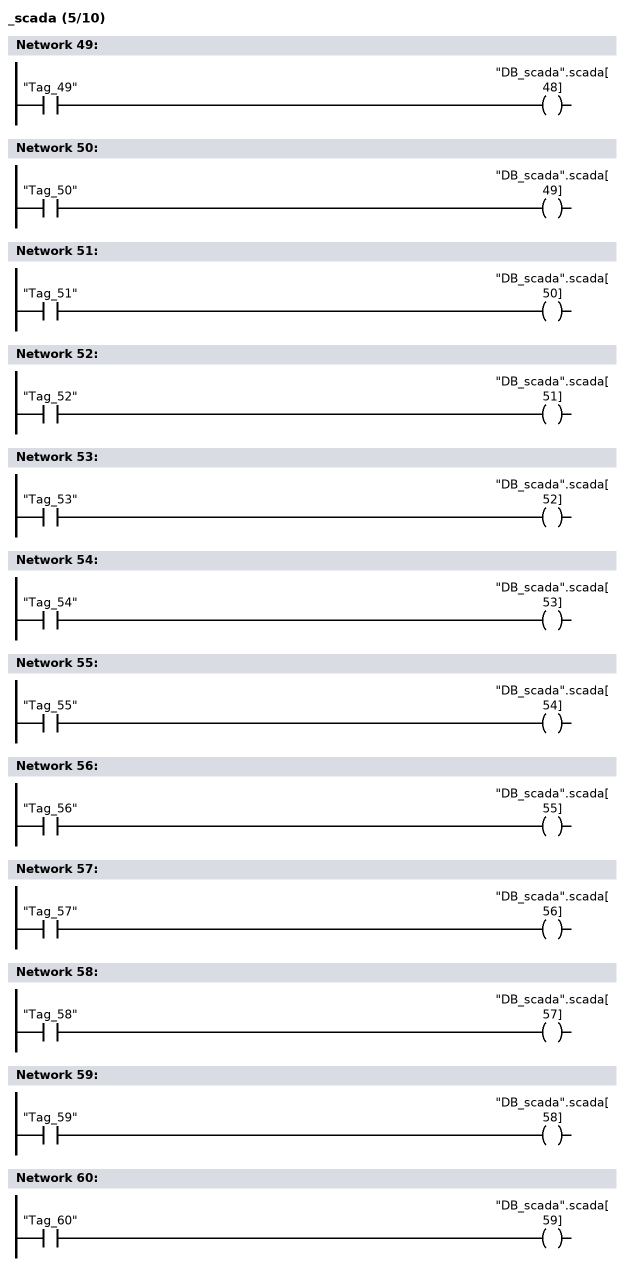
   RUNG wire#powerrail
      Contact( "Tag_49" )
      Coil( "DB_scada".scada[48] )
   END_RUNG
   // the same network as SCL:
   "DB_scada".scada[48] := "Tag_49";
END_REGION

REGION Network 50
   RUNG wire#powerrail
      Contact( "Tag_50" )
      Coil( "DB_scada".scada[49] )
   END_RUNG
   // the same network as SCL:
   "DB_scada".scada[49] := "Tag_50";
END_REGION

REGION Network 51
   RUNG wire#powerrail
      Contact( "Tag_51" )
      Coil( "DB_scada".scada[50] )
   END_RUNG
   // the same network as SCL:
   "DB_scada".scada[50] := "Tag_51";
END_REGION

REGION Network 52
   RUNG wire#powerrail
      Contact( "Tag_52" )
      Coil( "DB_scada".scada[51] )
   END_RUNG
   // the same network as SCL:
   "DB_scada".scada[51] := "Tag_52";
END_REGION

REGION Network 53
   RUNG wire#powerrail
      Contact( "Tag_53" )
      Coil( "DB_scada".scada[52] )
   END_RUNG
   // the same network as SCL:
   "DB_scada".scada[52] := "Tag_53";
END_REGION

REGION Network 54
   RUNG wire#powerrail
      Contact( "Tag_54" )
      Coil( "DB_scada".scada[53] )
   END_RUNG
   // the same network as SCL:
   "DB_scada".scada[53] := "Tag_54";
END_REGION

REGION Network 55
   RUNG wire#powerrail
      Contact( "Tag_55" )
      Coil( "DB_scada".scada[54] )
   END_RUNG
   // the same network as SCL:
   "DB_scada".scada[54] := "Tag_55";
END_REGION

REGION Network 56
   RUNG wire#powerrail
      Contact( "Tag_56" )
      Coil( "DB_scada".scada[55] )
   END_RUNG
   // the same network as SCL:
   "DB_scada".scada[55] := "Tag_56";
END_REGION

REGION Network 57
   RUNG wire#powerrail
      Contact( "Tag_57" )
      Coil( "DB_scada".scada[56] )
   END_RUNG
   // the same network as SCL:
   "DB_scada".scada[56] := "Tag_57";
END_REGION

REGION Network 58
   RUNG wire#powerrail
      Contact( "Tag_58" )
      Coil( "DB_scada".scada[57] )
   END_RUNG
   // the same network as SCL:
   "DB_scada".scada[57] := "Tag_58";
END_REGION

REGION Network 59
   RUNG wire#powerrail
      Contact( "Tag_59" )
      Coil( "DB_scada".scada[58] )
   END_RUNG
   // the same network as SCL:
   "DB_scada".scada[58] := "Tag_59";
END_REGION

REGION Network 60
   RUNG wire#powerrail
      Contact( "Tag_60" )
      Coil( "DB_scada".scada[59] )
   END_RUNG
   // the same network as SCL:
   "DB_scada".scada[59] := "Tag_60";
END_REGION

REGION Network 61
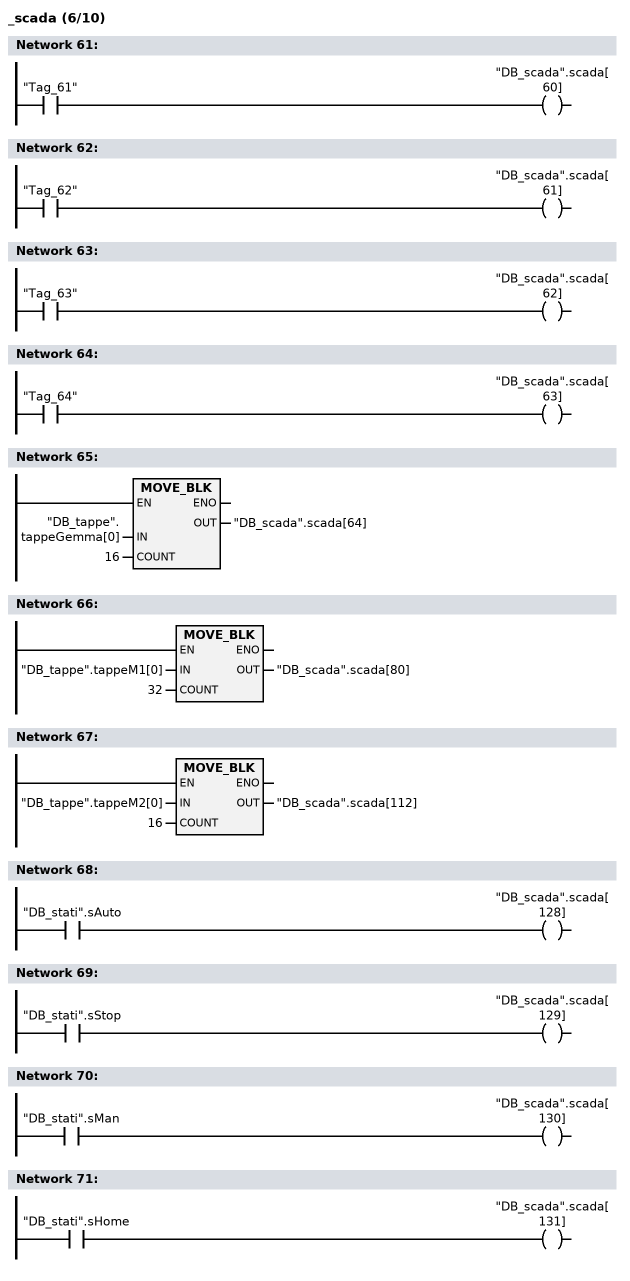
   RUNG wire#powerrail
      Contact( "Tag_61" )
      Coil( "DB_scada".scada[60] )
   END_RUNG
   // the same network as SCL:
   "DB_scada".scada[60] := "Tag_61";
END_REGION

REGION Network 62
   RUNG wire#powerrail
      Contact( "Tag_62" )
      Coil( "DB_scada".scada[61] )
   END_RUNG
   // the same network as SCL:
   "DB_scada".scada[61] := "Tag_62";
END_REGION

REGION Network 63
   RUNG wire#powerrail
      Contact( "Tag_63" )
      Coil( "DB_scada".scada[62] )
   END_RUNG
   // the same network as SCL:
   "DB_scada".scada[62] := "Tag_63";
END_REGION

REGION Network 64
   RUNG wire#powerrail
      Contact( "Tag_64" )
      Coil( "DB_scada".scada[63] )
   END_RUNG
   // the same network as SCL:
   "DB_scada".scada[63] := "Tag_64";
END_REGION

REGION Network 65
   MOVE_BLK(IN := "DB_tappe".tappeGemma[0], COUNT := 16, OUT => "DB_scada".scada[64]);
END_REGION

REGION Network 66
   MOVE_BLK(IN := "DB_tappe".tappeM1[0], COUNT := 32, OUT => "DB_scada".scada[80]);
END_REGION

REGION Network 67
   MOVE_BLK(IN := "DB_tappe".tappeM2[0], COUNT := 16, OUT => "DB_scada".scada[112]);
END_REGION

REGION Network 68
   RUNG wire#powerrail
      Contact( "DB_stati".sAuto )
      Coil( "DB_scada".scada[128] )
   END_RUNG
   // the same network as SCL:
   "DB_scada".scada[128] := "DB_stati".sAuto;
END_REGION

REGION Network 69
   RUNG wire#powerrail
      Contact( "DB_stati".sStop )
      Coil( "DB_scada".scada[129] )
   END_RUNG
   // the same network as SCL:
   "DB_scada".scada[129] := "DB_stati".sStop;
END_REGION

REGION Network 70
   RUNG wire#powerrail
      Contact( "DB_stati".sMan )
      Coil( "DB_scada".scada[130] )
   END_RUNG
   // the same network as SCL:
   "DB_scada".scada[130] := "DB_stati".sMan;
END_REGION

REGION Network 71
   RUNG wire#powerrail
      Contact( "DB_stati".sHome )
      Coil( "DB_scada".scada[131] )
   END_RUNG
   // the same network as SCL:
   "DB_scada".scada[131] := "DB_stati".sHome;
END_REGION

REGION Network 72
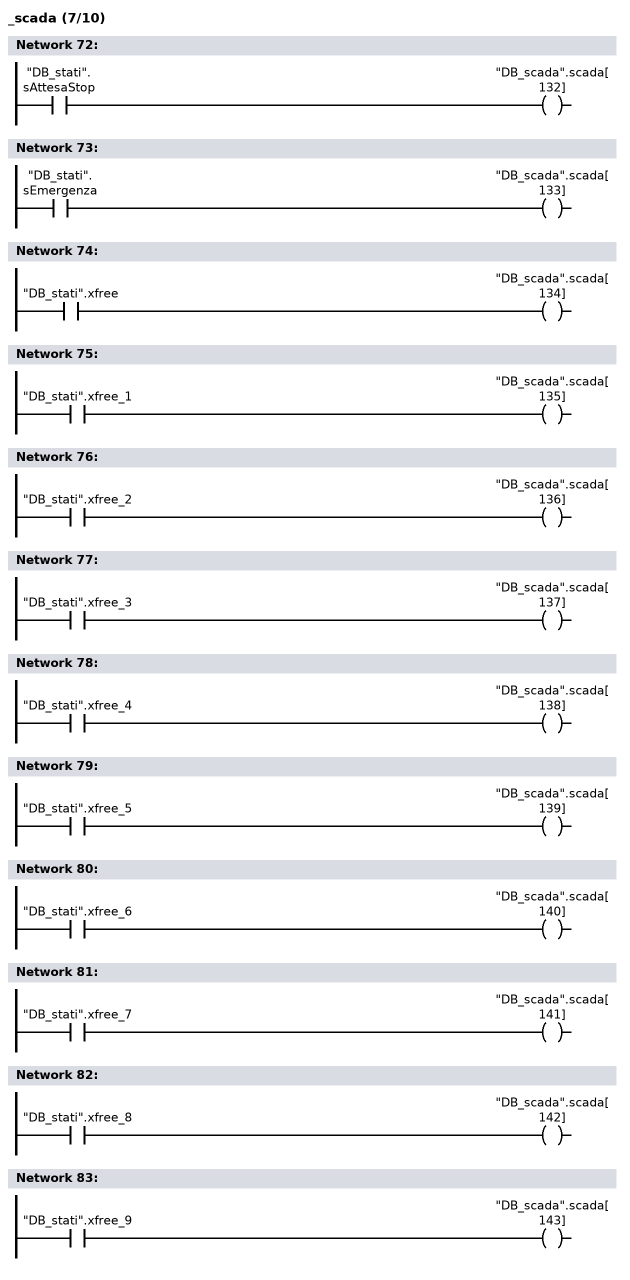
   RUNG wire#powerrail
      Contact( "DB_stati".sAttesaStop )
      Coil( "DB_scada".scada[132] )
   END_RUNG
   // the same network as SCL:
   "DB_scada".scada[132] := "DB_stati".sAttesaStop;
END_REGION

REGION Network 73
   RUNG wire#powerrail
      Contact( "DB_stati".sEmergenza )
      Coil( "DB_scada".scada[133] )
   END_RUNG
   // the same network as SCL:
   "DB_scada".scada[133] := "DB_stati".sEmergenza;
END_REGION

REGION Network 74
   RUNG wire#powerrail
      Contact( "DB_stati".xfree )
      Coil( "DB_scada".scada[134] )
   END_RUNG
   // the same network as SCL:
   "DB_scada".scada[134] := "DB_stati".xfree;
END_REGION

REGION Network 75
   RUNG wire#powerrail
      Contact( "DB_stati".xfree_1 )
      Coil( "DB_scada".scada[135] )
   END_RUNG
   // the same network as SCL:
   "DB_scada".scada[135] := "DB_stati".xfree_1;
END_REGION

REGION Network 76
   RUNG wire#powerrail
      Contact( "DB_stati".xfree_2 )
      Coil( "DB_scada".scada[136] )
   END_RUNG
   // the same network as SCL:
   "DB_scada".scada[136] := "DB_stati".xfree_2;
END_REGION

REGION Network 77
   RUNG wire#powerrail
      Contact( "DB_stati".xfree_3 )
      Coil( "DB_scada".scada[137] )
   END_RUNG
   // the same network as SCL:
   "DB_scada".scada[137] := "DB_stati".xfree_3;
END_REGION

REGION Network 78
   RUNG wire#powerrail
      Contact( "DB_stati".xfree_4 )
      Coil( "DB_scada".scada[138] )
   END_RUNG
   // the same network as SCL:
   "DB_scada".scada[138] := "DB_stati".xfree_4;
END_REGION

REGION Network 79
   RUNG wire#powerrail
      Contact( "DB_stati".xfree_5 )
      Coil( "DB_scada".scada[139] )
   END_RUNG
   // the same network as SCL:
   "DB_scada".scada[139] := "DB_stati".xfree_5;
END_REGION

REGION Network 80
   RUNG wire#powerrail
      Contact( "DB_stati".xfree_6 )
      Coil( "DB_scada".scada[140] )
   END_RUNG
   // the same network as SCL:
   "DB_scada".scada[140] := "DB_stati".xfree_6;
END_REGION

REGION Network 81
   RUNG wire#powerrail
      Contact( "DB_stati".xfree_7 )
      Coil( "DB_scada".scada[141] )
   END_RUNG
   // the same network as SCL:
   "DB_scada".scada[141] := "DB_stati".xfree_7;
END_REGION

REGION Network 82
   RUNG wire#powerrail
      Contact( "DB_stati".xfree_8 )
      Coil( "DB_scada".scada[142] )
   END_RUNG
   // the same network as SCL:
   "DB_scada".scada[142] := "DB_stati".xfree_8;
END_REGION

REGION Network 83
   RUNG wire#powerrail
      Contact( "DB_stati".xfree_9 )
      Coil( "DB_scada".scada[143] )
   END_RUNG
   // the same network as SCL:
   "DB_scada".scada[143] := "DB_stati".xfree_9;
END_REGION

REGION Network 84
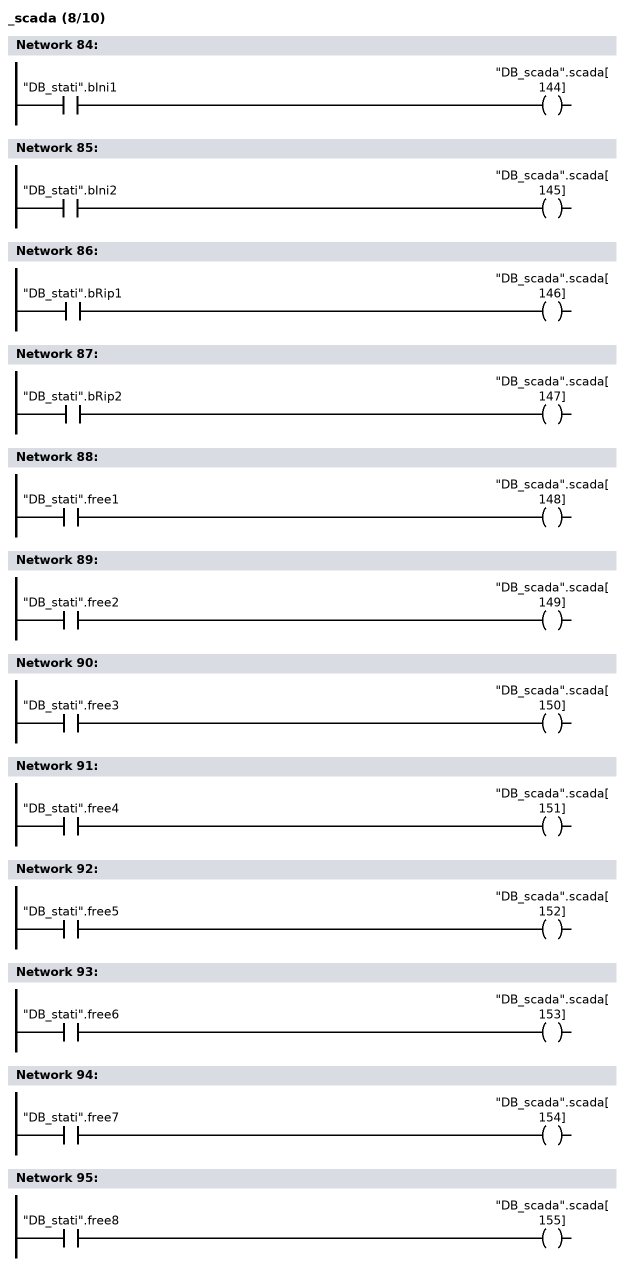
   RUNG wire#powerrail
      Contact( "DB_stati".bIni1 )
      Coil( "DB_scada".scada[144] )
   END_RUNG
   // the same network as SCL:
   "DB_scada".scada[144] := "DB_stati".bIni1;
END_REGION

REGION Network 85
   RUNG wire#powerrail
      Contact( "DB_stati".bIni2 )
      Coil( "DB_scada".scada[145] )
   END_RUNG
   // the same network as SCL:
   "DB_scada".scada[145] := "DB_stati".bIni2;
END_REGION

REGION Network 86
   RUNG wire#powerrail
      Contact( "DB_stati".bRip1 )
      Coil( "DB_scada".scada[146] )
   END_RUNG
   // the same network as SCL:
   "DB_scada".scada[146] := "DB_stati".bRip1;
END_REGION

REGION Network 87
   RUNG wire#powerrail
      Contact( "DB_stati".bRip2 )
      Coil( "DB_scada".scada[147] )
   END_RUNG
   // the same network as SCL:
   "DB_scada".scada[147] := "DB_stati".bRip2;
END_REGION

REGION Network 88
   RUNG wire#powerrail
      Contact( "DB_stati".free1 )
      Coil( "DB_scada".scada[148] )
   END_RUNG
   // the same network as SCL:
   "DB_scada".scada[148] := "DB_stati".free1;
END_REGION

REGION Network 89
   RUNG wire#powerrail
      Contact( "DB_stati".free2 )
      Coil( "DB_scada".scada[149] )
   END_RUNG
   // the same network as SCL:
   "DB_scada".scada[149] := "DB_stati".free2;
END_REGION

REGION Network 90
   RUNG wire#powerrail
      Contact( "DB_stati".free3 )
      Coil( "DB_scada".scada[150] )
   END_RUNG
   // the same network as SCL:
   "DB_scada".scada[150] := "DB_stati".free3;
END_REGION

REGION Network 91
   RUNG wire#powerrail
      Contact( "DB_stati".free4 )
      Coil( "DB_scada".scada[151] )
   END_RUNG
   // the same network as SCL:
   "DB_scada".scada[151] := "DB_stati".free4;
END_REGION

REGION Network 92
   RUNG wire#powerrail
      Contact( "DB_stati".free5 )
      Coil( "DB_scada".scada[152] )
   END_RUNG
   // the same network as SCL:
   "DB_scada".scada[152] := "DB_stati".free5;
END_REGION

REGION Network 93
   RUNG wire#powerrail
      Contact( "DB_stati".free6 )
      Coil( "DB_scada".scada[153] )
   END_RUNG
   // the same network as SCL:
   "DB_scada".scada[153] := "DB_stati".free6;
END_REGION

REGION Network 94
   RUNG wire#powerrail
      Contact( "DB_stati".free7 )
      Coil( "DB_scada".scada[154] )
   END_RUNG
   // the same network as SCL:
   "DB_scada".scada[154] := "DB_stati".free7;
END_REGION

REGION Network 95
   RUNG wire#powerrail
      Contact( "DB_stati".free8 )
      Coil( "DB_scada".scada[155] )
   END_RUNG
   // the same network as SCL:
   "DB_scada".scada[155] := "DB_stati".free8;
END_REGION

REGION Network 96
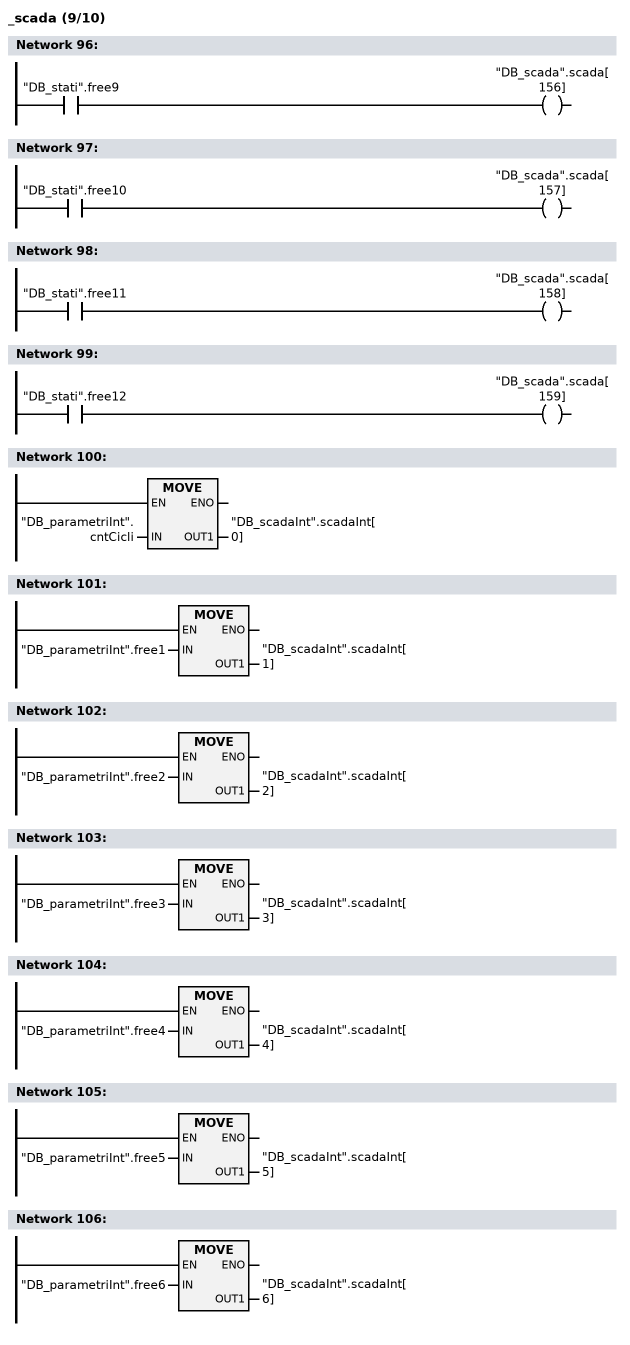
   RUNG wire#powerrail
      Contact( "DB_stati".free9 )
      Coil( "DB_scada".scada[156] )
   END_RUNG
   // the same network as SCL:
   "DB_scada".scada[156] := "DB_stati".free9;
END_REGION

REGION Network 97
   RUNG wire#powerrail
      Contact( "DB_stati".free10 )
      Coil( "DB_scada".scada[157] )
   END_RUNG
   // the same network as SCL:
   "DB_scada".scada[157] := "DB_stati".free10;
END_REGION

REGION Network 98
   RUNG wire#powerrail
      Contact( "DB_stati".free11 )
      Coil( "DB_scada".scada[158] )
   END_RUNG
   // the same network as SCL:
   "DB_scada".scada[158] := "DB_stati".free11;
END_REGION

REGION Network 99
   RUNG wire#powerrail
      Contact( "DB_stati".free12 )
      Coil( "DB_scada".scada[159] )
   END_RUNG
   // the same network as SCL:
   "DB_scada".scada[159] := "DB_stati".free12;
END_REGION

REGION Network 100
   RUNG wire#powerrail
      Move(in := "DB_parametriInt".cntCicli, out1 => "DB_scadaInt".scadaInt[0])
   END_RUNG
   // the same network as SCL:
   "DB_scadaInt".scadaInt[0] := "DB_parametriInt".cntCicli;
END_REGION

REGION Network 101
   RUNG wire#powerrail
      Move(in := "DB_parametriInt".free1, out1 => "DB_scadaInt".scadaInt[1])
   END_RUNG
   // the same network as SCL:
   "DB_scadaInt".scadaInt[1] := "DB_parametriInt".free1;
END_REGION

REGION Network 102
   RUNG wire#powerrail
      Move(in := "DB_parametriInt".free2, out1 => "DB_scadaInt".scadaInt[2])
   END_RUNG
   // the same network as SCL:
   "DB_scadaInt".scadaInt[2] := "DB_parametriInt".free2;
END_REGION

REGION Network 103
   RUNG wire#powerrail
      Move(in := "DB_parametriInt".free3, out1 => "DB_scadaInt".scadaInt[3])
   END_RUNG
   // the same network as SCL:
   "DB_scadaInt".scadaInt[3] := "DB_parametriInt".free3;
END_REGION

REGION Network 104
   RUNG wire#powerrail
      Move(in := "DB_parametriInt".free4, out1 => "DB_scadaInt".scadaInt[4])
   END_RUNG
   // the same network as SCL:
   "DB_scadaInt".scadaInt[4] := "DB_parametriInt".free4;
END_REGION

REGION Network 105
   RUNG wire#powerrail
      Move(in := "DB_parametriInt".free5, out1 => "DB_scadaInt".scadaInt[5])
   END_RUNG
   // the same network as SCL:
   "DB_scadaInt".scadaInt[5] := "DB_parametriInt".free5;
END_REGION

REGION Network 106
   RUNG wire#powerrail
      Move(in := "DB_parametriInt".free6, out1 => "DB_scadaInt".scadaInt[6])
   END_RUNG
   // the same network as SCL:
   "DB_scadaInt".scadaInt[6] := "DB_parametriInt".free6;
END_REGION

REGION Network 107
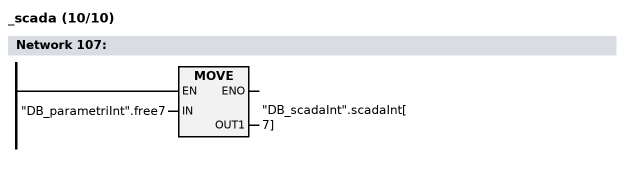
   RUNG wire#powerrail
      Move(in := "DB_parametriInt".free7, out1 => "DB_scadaInt".scadaInt[7])
   END_RUNG
   // the same network as SCL:
   "DB_scadaInt".scadaInt[7] := "DB_parametriInt".free7;
END_REGION
END_FUNCTION

ORGANIZATION_BLOCK "Main"   // OB1, LAD, ProgramCycle
TITLE = "Main Program Sweep (Cycle)"
{ S7_Optimized_Access := 'TRUE' }
VERSION : 0.1
   VAR_INPUT
      Initial_Call : Bool;   // Initial call of this OB
      Remanence : Bool;   // =True, if remanent data are available
   END_VAR
BEGIN

REGION Network 1
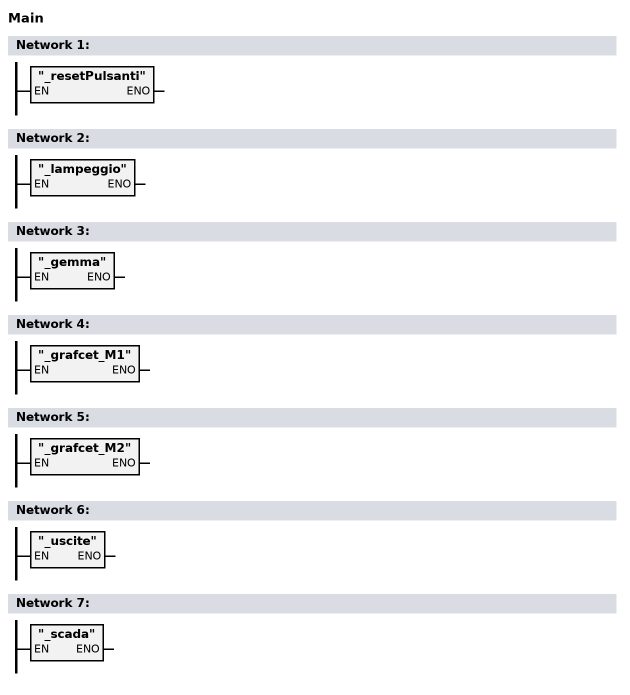
   RUNG wire#powerrail
      "_resetPulsanti"()
   END_RUNG
   // the same network as SCL:
   "_resetPulsanti"();
END_REGION

REGION Network 2
   RUNG wire#powerrail
      "_lampeggio"()
   END_RUNG
   // the same network as SCL:
   "_lampeggio"();
END_REGION

REGION Network 3
   RUNG wire#powerrail
      "_gemma"()
   END_RUNG
   // the same network as SCL:
   "_gemma"();
END_REGION

REGION Network 4
   RUNG wire#powerrail
      "_grafcet_M1"()
   END_RUNG
   // the same network as SCL:
   "_grafcet_M1"();
END_REGION

REGION Network 5
   RUNG wire#powerrail
      "_grafcet_M2"()
   END_RUNG
   // the same network as SCL:
   "_grafcet_M2"();
END_REGION

REGION Network 6
   RUNG wire#powerrail
      "_uscite"()
   END_RUNG
   // the same network as SCL:
   "_uscite"();
END_REGION

REGION Network 7
   RUNG wire#powerrail
      "_scada"()
   END_RUNG
   // the same network as SCL:
   "_scada"();
END_REGION
END_ORGANIZATION_BLOCK